Staubli VAL3: BalayageSimple.pgx

program BalayageSimple()
begin
  //Rappel : pInitialPosition = {{597.67, 50, -72.68,-180,0,-180}, {sfree, efree, wfree}}
  while bAcquisitionStarted == false
  endWhile

  pNextPosition = pInitialPosition
    for nNextPositionX = pInitialPosition.trsf.x - nScanningLength/2 to pInitialPosition.trsf.x + nScanningLength/2 step nScanningLength / nScanningLineNumber
      pNextPosition.trsf.y = pInitialPosition.trsf.y - nScanningWidth/2
      pNextPosition.trsf.x = nNextPositionX
      movel(pNextPosition, flange, mNomSpeed)
      waitEndMove()
      pNextPosition.trsf.y = pInitialPosition.trsf.y + nScanningWidth/2
      movel(pNextPosition, flange, mNomSpeed)
      waitEndMove()
    endFor
    pNextPosition.trsf.x = pInitialPosition.trsf.x
    pNextPosition.trsf.y = pInitialPosition.trsf.y - nScanningWidth/2
    movec(pCircle,pNextPosition,flange,mNomSpeed)
    waitEndMove()
end
